// TIA Portal V18 export
VAR_GLOBAL   // PLC tag table "Cabinet_4"
   Sz4_Button_LED_ST32_ST33 AT %Q1400.0 : Bool;
   Sz4_Button_LED_ST33_ST34 AT %Q1400.1 : Bool;
   Sz4_Button_LED_ST36_ST38 AT %Q1400.2 : Bool;
   Sz4_Button_LED_ST37_ST36 AT %Q1400.3 : Bool;
   Sz4_Button_LED_ST34_ST33 AT %Q1400.4 : Bool;
   Sz4_Button_LED_ST38_ST36 AT %Q1400.5 : Bool;
   "Reserved(58)" AT %Q1400.6 : Bool;
   "Reserved(59)" AT %Q1400.7 : Bool;
   Sz4_ST32_SenA AT %I1400.0 : Bool;
   Sz4_ST32_SenB AT %I1400.1 : Bool;
   Sz4_ST32_SenC AT %I1400.2 : Bool;
   Sz4_ST32_SenD AT %I1400.3 : Bool;
   Sz4_ST33_SenA AT %I1400.4 : Bool;
   Sz4_ST33_SenB AT %I1400.5 : Bool;
   Sz4_ST33_SenC AT %I1400.6 : Bool;
   Sz4_ST33_SenD AT %I1400.7 : Bool;
   Sz4_ST36_SenA AT %I1401.0 : Bool;
   Sz4_ST36_SenB AT %I1401.1 : Bool;
   Sz4_ST36_SenC AT %I1401.2 : Bool;
   Sz4_ST36_SenD AT %I1401.3 : Bool;
   Sz4_ST37_SenA AT %I1401.4 : Bool;
   Sz4_ST37_SenB AT %I1401.5 : Bool;
   Sz4_ST37_SenC AT %I1401.6 : Bool;
   Sz4_ST37_SenD AT %I1401.7 : Bool;
   Sz4_Button_ST32_ST33 AT %I1402.0 : Bool;
   Sz4_Button_ST33_ST34 AT %I1402.1 : Bool;
   Sz4_Button_ST36_ST38 AT %I1402.2 : Bool;
   Sz4_Button_ST37_ST36 AT %I1402.3 : Bool;
   Sz4_Button_ST34_ST33 AT %I1402.4 : Bool;
   Sz4_Button_ST38_ST36 AT %I1402.5 : Bool;
   "Reserved(60)" AT %I1402.6 : Bool;
   "Reserved(61)" AT %I1402.7 : Bool;
   Sz4_Safety1_1 AT %I1403.0 : Bool;
   "Reserved(62)" AT %I1403.1 : Bool;
   "Reserved(63)" AT %I1403.2 : Bool;
   "Reserved(64)" AT %I1403.3 : Bool;
   Sz4_Safety1_2 AT %I1403.4 : Bool;
   "Reserved(65)" AT %I1403.5 : Bool;
   "Reserved(66)" AT %I1403.6 : Bool;
   "Reserved(67)" AT %I1403.7 : Bool;
   "Reserved(75)" AT %I1404.0 : Bool;
   "Reserved(74)" AT %I1404.1 : Bool;
   "Reserved(73)" AT %I1404.2 : Bool;
   "Reserved(72)" AT %I1404.3 : Bool;
   "Reserved(71)" AT %I1404.4 : Bool;
   "Reserved(70)" AT %I1404.5 : Bool;
   "Reserved(69)" AT %I1404.6 : Bool;
   "Reserved(68)" AT %I1404.7 : Bool;
END_VAR
